Universal Robots PolyScope program: Test Program.urp

Program Test Program (installation=default directory=/home/ur3simulator/Downloads/ursim-3.12.1.90940/programs/Test Program createdIn=3.12.1.90940 lastSavedIn=3.12.1.90940 robotSerialNumber=2018339999)
Calibrated DH parameters: a=[0, -0.24365, -0.21325, 0, 0, 0]; d=[0.1519, 0, 0, 0.11235, 0.08535, 0.0819]; alpha=[1.570796, 0, 0, 1.570796, -1.570796, 0]; deltaTheta=[0, 0, 0, 0, 0, 0]
InitVariablesNode variables(variable(name=cnt_1, expression=0))
Robot Program (runOnlyOnce=false)
  Pallet pattern(dimensionality=List firstAxisCount=5 secondAxisCount=5 thirdAxisCount=5 motionType=MoveL speed=0.25 acceleration=1.2 useActiveTCP=true, counterVariable(name=cnt_1, initializeExpression=0), patternPoseVariable(name=pose_1), feature=Base, children(Waypoint(type=Fixed name=Waypoint_1, position(joints=-1.927315009747642, -1.9188016317747874, -1.9332272964740707, -0.8925078079375481, 1.5855677274552349, -0.3575397577849291 pose=-0.21842707618624274, -0.2680453239215242, 0.1572781598013413, -0.0012212120504216239, 3.1162764576489637, 0.038892054509567085), poseInFeatureCoordinates=[-0.218427, -0.268045, 0.157278, -0.001221, 3.116276, 0.038892], outputFlangePose=[-0.218427, -0.268045, 0.157278, -0.001221, 3.116276, 0.038892]), Waypoint(type=Fixed name=Waypoint_2, position(joints=-2.1276149037920966, -2.1122903403855418, -1.619208074207723, -1.0153336079920372, 1.5788775105216057, -0.5577415253651381 pose=-0.29842704051674807, -0.26804535113871025, 0.15727819922446767, -0.0012212827746720994, 3.116276507089661, 0.03889177753061143), poseInFeatureCoordinates=[-0.298427, -0.268045, 0.157278, -0.001221, 3.116277, 0.038892], outputFlangePose=[-0.298427, -0.268045, 0.157278, -0.001221, 3.116276, 0.038892]), Waypoint(type=Fixed name=Waypoint_3, position(joints=-2.2464849976401755, -2.2843709669050183, -1.313598157377652, -1.1495776523695689, 1.574736809626445, -0.6765417561610905 pose=-0.358427090910527, -0.26804536901564796, 0.15727826655924093, -0.001220992721180084, 3.116276739499061, 0.038891284273906236), poseInFeatureCoordinates=[-0.358427, -0.268045, 0.157278, -0.001221, 3.116277, 0.038891], outputFlangePose=[-0.358427, -0.268045, 0.157278, -0.001221, 3.116277, 0.038892]))); actionSequence(name=PalletSequence motionType=MoveL speed=0.25 acceleration=1.2 useActiveTCP=true, anchorWaypoint(type=Fixed name=PatternPoint_1, position(joints=-2.2464849976401755, -2.2843709669050183, -1.313598157377652, -1.1495776523695689, 1.574736809626445, -0.6765417561610905 pose=-0.358427090910527, -0.26804536901564796, 0.15727826655924093, -0.001220992721180084, 3.116276739499061, 0.038891284273906236), poseInFeatureCoordinates=[-0.358427, -0.268045, 0.157278, -0.001221, 3.116277, 0.038891], outputFlangePose=[-0.358427, -0.268045, 0.157278, -0.001221, 3.116277, 0.038892]), feature=Base, children(Waypoint(type=Fixed name=Waypoint_4, position(joints=-1.9273150602837292, -1.7012121018846607, -1.4820752844378902, -1.5612494426548915, 1.5855675935751703, -0.35753995576266817 pose=-0.2184271254573415, -0.2680454281619303, 0.2999998571683863, -0.0012212095223541114, 3.1162763932485347, 0.03889281493098355), poseInFeatureCoordinates=[-0.218427, -0.268045, 0.3, -0.001221, 3.116276, 0.038893], outputFlangePose=[-0.218427, -0.268045, 0.3, -0.001221, 3.116277, 0.038892]), Waypoint(type=Fixed name=Approach_1, motionParameters(nextMotionTime=2), position(joints=-2.2464850583942404, -2.1846425578709585, -0.7978748389762798, -1.7650289898553382, 1.574736833574871, -0.6765416303547003 pose=-0.35842711035821256, -0.26804539323127424, 0.3000000171579963, -0.001220993513208907, 3.1162768922805264, 0.0388909963259509), poseInFeatureCoordinates=[-0.358427, -0.268045, 0.3, -0.001221, 3.116277, 0.038891], outputFlangePose=[-0.358427, -0.268045, 0.3, -0.001221, 3.116277, 0.038891]), Waypoint=PatternPoint_1, Set(type=NoAction), Wait(type=Sleep, waitTime=0.01), Waypoint(type=Fixed name=Exit_1, position(joints=-2.2464849976401755, -2.2843709669050183, -1.313598157377652, -1.1495776523695689, 1.574736809626445, -0.6765417561610905 pose=-0.358427090910527, -0.26804536901564796, 0.15727826655924093, -0.001220992721180084, 3.116276739499061, 0.038891284273906236), poseInFeatureCoordinates=[-0.358427, -0.268045, 0.157278, -0.001221, 3.116277, 0.038891], outputFlangePose=[-0.358427, -0.268045, 0.157278, -0.001221, 3.116277, 0.038892])))
    Pattern -> pattern
    AnchoredSequence -> PalletSequence
